Fanuc KAREL source: ROUND.kl

PROGRAM T
%NOLOCKGROUP
VAR
 v0 : REAL
 res : INTEGER
BEGIN
 res = ROUND(v0)
END T
